// TIA Portal project "Elevator" (V14)

(* hardware
DEVICE "S7-1200 station_1"  S7-1200 Station
   slot 0: "Rack_0"  Rack  V1.0
   slot 1: "PLC_1"  Unspecific CPU 1200  6ES7 2XX-XXXXX-XXXX  V4.2
*)

// ===== PLC "PLC_1"  Unspecific CPU 1200 =====

VAR_GLOBAL   // PLC tag table "Default tag table"
   "DI_btnCall0KuEn" AT %I0.0 : Bool;   // knop verdieping 0, lift aanroepen
   "DI_btnCall1KuEn" AT %I0.1 : Bool;   // knop verdieping 1, lift aanroepen
   "DI_btnCall2KuEn" AT %I0.2 : Bool;   // knop verdieping 2, lift aanroepen
   "DI_btnElev0KuEn" AT %I0.3 : Bool;   // knop in de lift, gaat naar verdieping 0
   "DI_btnElev1KuEn" AT %I0.4 : Bool;   // knop in de lift, gaat naar verdieping 1
   "DI_btnElev2KuEn" AT %I0.5 : Bool;   // knop in de lift, gaat naar verdieping 2
   "DI_eleFloor0KuEn" AT %I0.6 : Bool;   // True, als de lift op verdieping 0 is
   "DI_eleFloor1KuEn" AT %I0.7 : Bool;   // True, als de lift op verdieping 1 is
   "DI_eleFloor2KuEn" AT %I1.0 : Bool;   // True, als de lift op verdieping 2 is
   "DI_doorClosed0KuEn" AT %I1.1 : Bool;   // True, als deur op verdieping 0 is gesloten
   "DI_doorClosed1KuEn" AT %I1.2 : Bool;   // True, als deur op verdieping 1 is gesloten
   "DI_doorClosed2KuEn" AT %I1.3 : Bool;   // True, als deur op verdieping 2 is gesloten
   "DQ_motorUpKuEn" AT %Q0.0 : Bool;   // Lift gaat naar boven als het True is.
   "DQ_motorDownKuEn" AT %Q0.1 : Bool;   // Lift gaat naar onder als het True is.
   "DQ_openDoor0KuEn" AT %Q0.2 : Bool;   // Deur op verdieping 0 gaat open als het True is.
   "DQ_openDoor1KuEn" AT %Q0.3 : Bool;   // Deur op verdieping 1 gaat open als het True is.
   "DQ_openDoor2KuEn" AT %Q0.4 : Bool;   // Deur op verdieping 2 gaat open als het True is.
END_VAR

FUNCTION "blcMain" : Void   // FC1, SCL
{ S7_Optimized_Access := 'TRUE' }
VERSION : 0.1
BEGIN
   (*trigButtonsKusD(CLK:= xBtnOnOffKusD OR xBtnMenuKusD, Q=> xPulseKusD);*)

   IF "DI_btnCall0KuEn" = TRUE OR "DI_btnElev0KuEn" THEN

       //De motor moet uit staan
       IF "DQ_motorUpKuEn" = FALSE AND "DQ_motorDownKuEn" = FALSE THEN

           //Als de lift op de begane grond staat:
           IF "DI_eleFloor0KuEn" = TRUE THEN
               "DQ_openDoor0KuEn" := TRUE;//Deur gaat open
           END_IF;

           //Als de lift op de 1ste of 2de verdieping staat:
           IF "DI_eleFloor1KuEn" = TRUE OR "DI_eleFloor2KuEn" = TRUE THEN
               "DQ_openDoor1KuEn" := FALSE;
               "DQ_openDoor2KuEn" := FALSE;
               "DQ_motorDownKuEn" := TRUE;//Motor gaat naar benenden

               //Motor zal naar beneden gaan tot dat de lift op de begane grond staat.
               WHILE "DQ_motorDownKuEn" = TRUE DO
                   IF "DI_eleFloor0KuEn" = TRUE THEN
                       "DQ_motorDownKuEn" := FALSE;
                       "DQ_openDoor0KuEn" := TRUE;
                   END_IF;
               END_WHILE;
           END_IF;
       ELSE
           ;
       END_IF;

   END_IF;

   IF "DI_btnCall1KuEn" = TRUE OR "DI_btnElev1KuEn" THEN

       IF "DQ_motorUpKuEn" = FALSE AND "DQ_motorDownKuEn" = FALSE THEN

           IF "DI_eleFloor0KuEn" = TRUE THEN
               "DQ_openDoor0KuEn" := FALSE;
               "DQ_motorUpKuEn" := TRUE;

               WHILE "DQ_motorUpKuEn" = TRUE DO
                   IF "DI_eleFloor1KuEn" = TRUE THEN
                       "DQ_motorUpKuEn" := FALSE;
                       "DQ_openDoor1KuEn" := TRUE;
                   END_IF;
               END_WHILE;
           END_IF;

           IF "DI_eleFloor1KuEn" = TRUE THEN
               "DQ_openDoor1KuEn" := TRUE;
           END_IF;

           IF "DI_eleFloor2KuEn" = TRUE THEN
               "DQ_openDoor2KuEn" := FALSE;
               "DQ_motorDownKuEn" := TRUE;

               WHILE "DQ_motorDownKuEn" = TRUE DO
                   IF "DI_eleFloor1KuEn" = TRUE THEN
                       "DQ_motorDownKuEn" := FALSE;
                       "DQ_openDoor1KuEn" := TRUE;
                   END_IF;
               END_WHILE;
           END_IF;

       ELSE
           ;
       END_IF;

   END_IF;

   IF "DI_btnCall2KuEn" = TRUE OR "DI_btnElev2KuEn" THEN

       IF "DQ_motorUpKuEn" = FALSE AND "DQ_motorDownKuEn" = FALSE THEN

           IF "DI_eleFloor0KuEn" = TRUE OR "DI_eleFloor1KuEn" = TRUE THEN
               "DQ_openDoor0KuEn" := FALSE;
               "DQ_openDoor1KuEn" := FALSE;
               "DQ_motorUpKuEn" := TRUE;

               WHILE "DQ_motorUpKuEn" = TRUE DO
                   IF "DI_eleFloor2KuEn" = TRUE THEN
                       "DQ_motorUpKuEn" := FALSE;
                       "DQ_openDoor2KuEn" := TRUE;
                   END_IF;
               END_WHILE;
           END_IF;

           IF "DI_eleFloor2KuEn" = TRUE THEN
               "DQ_openDoor2KuEn" := TRUE;
           END_IF;
       ELSE
           ;
       END_IF;

   END_IF;
END_FUNCTION

ORGANIZATION_BLOCK "Main"   // OB1, LAD, ProgramCycle
TITLE = "Main Program Sweep (Cycle)"
{ S7_Optimized_Access := 'TRUE' }
VERSION : 0.1
   VAR_INPUT
      Initial_Call : Bool;   // Initial call of this OB
      Remanence : Bool;   // =True, if remanent data are available
   END_VAR
BEGIN

REGION Network 1
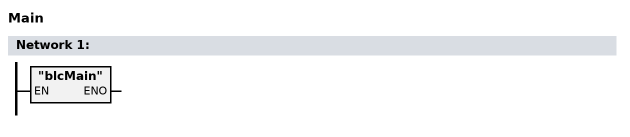
   RUNG wire#powerrail
      "blcMain"()
   END_RUNG
   // the same network as SCL:
   "blcMain"();
END_REGION
END_ORGANIZATION_BLOCK